# EPICS substitutions: iocBoot/gasFlowCalc.substitutions
file "./gasFlowCalc.db"
{
pattern
{Ch, DevIn, DevOut, ChOut, EGUF}
{1,  IO:1,  IO:2,   1,     100 }
{2,  IO:1,  IO:2,   2,     50 }
{3,  IO:1,  IO:2,   3,     50 }
{4,  IO:1,  IO:2,   4,     500 }
{5,  IO:1,  IO:3,   1,     50 }
{6,  IO:1,  IO:3,   2,     500 }
{7,  IO:1,  IO:3,   3,     50 }
{8,  IO:1,  IO:3,   4,     50 }
}
